KUKA KRL data list: Up206.dat

&ACCESS RVP
&REL 27
&COMMENT TCP Check Klebepistole
&PARAM EDITMASK = Up999[1-999]
&PARAM TEMPLATE = C:\KRC\Roboter\Template\upvorgabe
&PARAM TPVW_VERSION = 8.3.18
&PARAM DISKPATH = UPs
DEFDAT  Up206
; FOLD ;%{H} %MKUKATPVW
; ENDFOLD
; interface to basic routines
EXT  BAS (BAS_COMMAND  :IN,REAL  :IN )
; interface to VW-standard routines
EXT  VW (VW_COMMAND  :IN,BOOL  :IN,REAL  :IN,REAL  :IN,REAL  :IN,REAL  :IN,BOOL  :IN,E6POS  :IN )
; interface to VW_USER - Call
EXT  VW_USER (VW_USER_CMD  :IN,INT  :IN,REAL  :IN,REAL  :IN,REAL  :IN,REAL  :IN,REAL  :IN,REAL  :IN,REAL  :IN,REAL  :IN,REAL  :IN,BOOL  :IN )
EXT  VW_USR_R (VW_USER_CMD  :IN,INT  :IN,REAL  :IN,REAL  :IN,REAL  :IN,REAL  :IN,REAL  :IN,REAL  :IN,REAL  :IN,REAL  :IN,REAL  :IN,BOOL  :IN )
EXT  IBGN (IBGN_COMMAND  :IN,BOOL  :IN,REAL  :IN,REAL  :IN,BOOL  :IN,E6POS  :OUT )
; interface select routine
EXTFCT  INT  SELECT(SUBTYPE  :IN,INT  :IN,BOOL  :IN,ARI_TYP  :IN,INT  :IN,BOOL_TYP  :IN,INT  :IN,BOOL  :IN)
INT VW_NEXT_FREE=8
INT VW_NFREE_SPS=8
INT VW_MAX_SPS=108
DECL VW_MPARA_TYP P1_D={TOOL_NO 1,BASE_NO 0,VB 100,VE 0,ACC 100,TRG_TIME 0,MOVE_TYPE #PTP_MOTION}
DECL E6POS P1={X 97.7330475,Y 757.255310,Z 271.002808,A 0.0,B 90.0000,C 150.000,S 2,T 3,E1 0.0,E2 0.0,E3 0.0,E4 0.0,E5 0.0,E6 0.0}
DECL VW_MPARA_TYP P2_D={TOOL_NO 1,BASE_NO 0,VB 100,VE 100,ACC 100,TRG_TIME 0,MOVE_TYPE #PTP_MOTION}
DECL E6POS P2={X 149.655106,Y 750.154724,Z 71.1661911,A 115.568604,B 87.6566772,C -86.1345367,S 2,T 11,E1 0.0,E2 0.0,E3 0.0,E4 0.0,E5 0.0,E6 0.0}
DECL VW_MPARA_TYP P3_D={TOOL_NO 1,BASE_NO 0,VB 100,VE 100,ACC 100,TRG_TIME 0,MOVE_TYPE #PTP_MOTION}
DECL E6POS P3={X 149.334106,Y 571.239075,Z 86.8882599,A 7.28258514,B 89.4302292,C 165.599,S 2,T 3,E1 0.0,E2 0.0,E3 0.0,E4 0.0,E5 0.0,E6 0.0}
DECL VW_MPARA_TYP P4_D={TOOL_NO 1,BASE_NO 0,VB 250,VE 0,ACC 100,TRG_TIME 5,MOVE_TYPE #PATH_MOTION}
DECL E6POS P4={X 149.334106,Y 571.239075,Z 47.0881805,A 7.28258419,B 89.4302292,C 165.599,S 2,T 3,E1 0.0,E2 0.0,E3 0.0,E4 0.0,E5 0.0,E6 0.0}
DECL VW_MPARA_TYP P5_D={TOOL_NO 1,BASE_NO 0,VB 250,VE 100,ACC 100,TRG_TIME 0,MOVE_TYPE #PATH_MOTION}
DECL E6POS P5={X 149.334106,Y 571.239075,Z 86.8882599,A 7.28258514,B 89.4302292,C 165.599,S 2,T 3,E1 0.0,E2 0.0,E3 0.0,E4 0.0,E5 0.0,E6 0.0}
DECL VW_MPARA_TYP P6_D={TOOL_NO 1,BASE_NO 0,VB 100,VE 100,ACC 100,TRG_TIME 0,MOVE_TYPE #PTP_MOTION}
DECL E6POS P6={X 149.655106,Y 750.154724,Z 71.1661911,A 115.568604,B 87.6566772,C -86.1345367,S 2,T 11,E1 0.0,E2 0.0,E3 0.0,E4 0.0,E5 0.0,E6 0.0}
DECL VW_MPARA_TYP P7_D={TOOL_NO 1,BASE_NO 0,VB 100,VE 0,ACC 100,TRG_TIME 0,MOVE_TYPE #PTP_MOTION}
DECL E6POS P7={X 97.7330475,Y 757.255310,Z 271.002808,A 0.0,B 90.0000,C 150.000,S 2,T 3,E1 0.0,E2 0.0,E3 0.0,E4 0.0,E5 0.0,E6 0.0}
ENDDAT
